{attribute 'GeneratedUsingTerminal: KL2641'}
{attribute addProperty BoxType "KL2641"}
{attribute addProperty Id "StateAT %I*BOOL0OutputAT %Q*BOOL0"}
{attribute addProperty CRC "629786844"}
{attribute addProperty Size "0"}
TYPE Channel_2589C8DC :
STRUCT
	{attribute addProperty Name "State"}
	State AT %I* : BOOL;
	{attribute addProperty Name "Output"}
	Output AT %Q* : BOOL;
END_STRUCT
END_TYPE

(* stored: Version 1.2.0.0, ProductVersion 3.1.4024.9
   DUT Channel_2589C8DC: Id {f045db6f-9522-4577-b293-8876eed8a285} *)
